# EPICS substitutions: db/EL4032.substitutions
file EL4032.template
{ 	pattern
	{
		TERMINAL,
		DESC1,	SCAN1,	ADEL1,	EGUF1,	EGUL1,	DRVH1,	DRVL1,	HOPR1,	LOPR1,	LOLO1,	LOPR1,	PINI1,
		DESC2,	SCAN2,	ADEL2,	EGUF2,	EGUL2,	DRVH2,	DRVL2,	HOPR2,	LOPR2,	LOLO2,	LOPR2,	PINI2
	}
	{
	}
}
